FUNCTION_BLOCK LINKPUBLISHER (* Service Interface Function Block Type *)
  (* Standard: 61499-2 *)
  (* Version 0.0, 9/14/2008, Horst Mayer, nxtControl GmbH, template *)
  PACKAGE IEC61499;
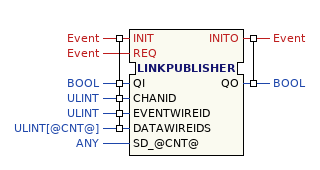
  EVENT_INPUT
    INIT WITH QI, CHANID, EVENTWIREID, DATAWIREIDS;
    REQ;
  END_EVENT
  EVENT_OUTPUT
    INITO WITH QO;
  END_EVENT
  VAR_INPUT
    QI : BOOL;
    CHANID : ULINT;
    EVENTWIREID : ULINT;
    DATAWIREIDS : ARRAY [@CNT@] OF ULINT;
    SD_@CNT@ : ANY;
  END_VAR
  VAR_OUTPUT
    QO : BOOL; (* Event Output Qualifier *)
  END_VAR
END_FUNCTION_BLOCK
